// SIMATIC STEP 7 (V5.x) project Simatic_Manager_HMI_Int
// CPU: CPU 315-2 DP
// station: Hardware
// station: SIMATIC 300(1)
// station: P_ADR_BUS
// station: P_ADR_BUS
// station: Configuration
// station: P_ADR_BUS
// station: Configuration
// program: S7 Program(1)

SYMBOL_TABLE
"ADD"	DB 1	DB 1
"VAT_1"	VAT 1	
END_SYMBOL_TABLE

DATA_BLOCK "ADD"	// DB 1
VERSION : 0.1
  STRUCT
   Start : BOOL ;	//Temporary placeholder variable
   Stop : BOOL ;
   Motor : BOOL ;
   SP_Temp : REAL ;
   PV_Temp : REAL ;
   SP_ADD1 : INT ;
   SP_ADD2 : INT ;
   SUM : INT ;
   MUL : INT ;
   SUB : INT ;
   DIV : INT ;
   SP1 : WORD ;
   SP2 : WORD ;
   SUM1 : WORD ;
  END_STRUCT ;	
BEGIN
END_DATA_BLOCK

ORGANIZATION_BLOCK OB 1
TITLE = "Main Program Sweep (Cycle)"
VERSION : 0.1
VAR_TEMP
  OB1_EV_CLASS : BYTE ;	//Bits 0-3 = 1 (Coming event), Bits 4-7 = 1 (Event class 1)
  OB1_SCAN_1 : BYTE ;	//1 (Cold restart scan 1 of OB 1), 3 (Scan 2-n of OB 1)
  OB1_PRIORITY : BYTE ;	//Priority of OB Execution
  OB1_OB_NUMBR : BYTE ;	//1 (Organization block 1, OB1)
  OB1_RESERVED_1 : BYTE ;	//Reserved for system
  OB1_RESERVED_2 : BYTE ;	//Reserved for system
  OB1_PREV_CYCLE : INT ;	//Cycle time of previous OB1 scan (milliseconds)
  OB1_MIN_CYCLE : INT ;	//Minimum cycle time of OB1 (milliseconds)
  OB1_MAX_CYCLE : INT ;	//Maximum cycle time of OB1 (milliseconds)
  OB1_DATE_TIME : DATE_AND_TIME ;	//Date and time OB1 started
END_VAR
BEGIN
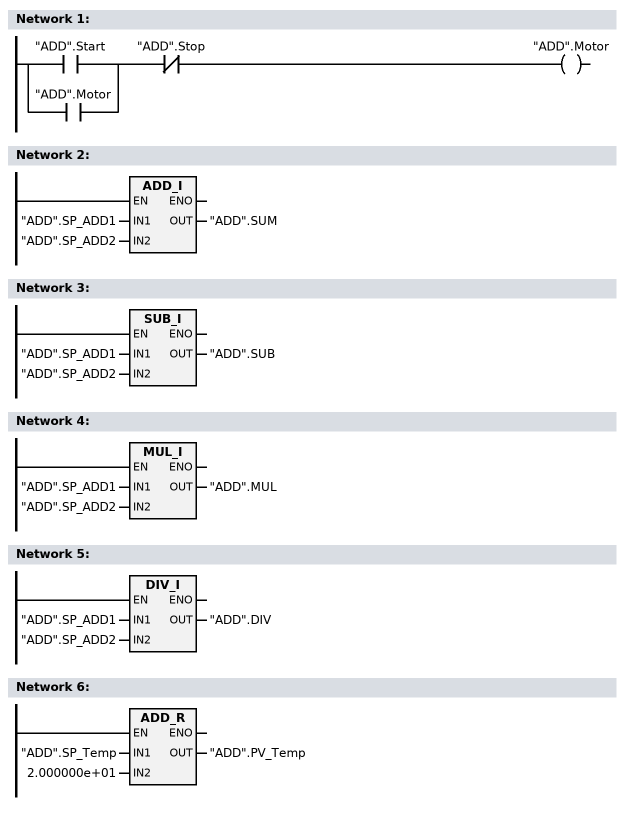
NETWORK
TITLE =
      A(;
      O     "ADD".Start;
      O     "ADD".Motor;
      );
      AN    "ADD".Stop;
      =     "ADD".Motor;
NETWORK
TITLE =
      L     "ADD".SP_ADD1;
      L     "ADD".SP_ADD2;
      +I;
      T     "ADD".SUM;
      NOP   0;
NETWORK
TITLE =
      L     "ADD".SP_ADD1;
      L     "ADD".SP_ADD2;
      -I;
      T     "ADD".SUB;
      NOP   0;
NETWORK
TITLE =
      L     "ADD".SP_ADD1;
      L     "ADD".SP_ADD2;
      *I;
      T     "ADD".MUL;
      NOP   0;
NETWORK
TITLE =
      L     "ADD".SP_ADD1;
      L     "ADD".SP_ADD2;
      /I;
      T     "ADD".DIV;
      NOP   0;
NETWORK
TITLE =
      L     "ADD".SP_Temp;
      L     2.000000e+01;
      +R;
      T     "ADD".PV_Temp;
      NOP   0;
END_ORGANIZATION_BLOCK
